{attribute 'linkalways'} 
{attribute 'no_explicit_call' := 'This FB is a CLASS and must be accessed using methods or properties'}
{attribute 'enable_dynamic_creation'}
FUNCTION_BLOCK Node_F_VN_MedianElementElementwise_TcVnPoint2_LREAL EXTENDS VisionNode
VAR
    ipContainer : _ITcVnContainer;
    aMedian : _TcVnPoint2_LREAL;
    hrPrev : _HRESULT(S_OK);
    hresult : _HRESULT(S_OK);
END_VAR

METHOD PUBLIC  Clone : I_Node
VAR
	pNode : POINTER TO Node_F_VN_MedianElementElementwise_TcVnPoint2_LREAL;
END_VAR
pNode := __NEW(Node_F_VN_MedianElementElementwise_TcVnPoint2_LREAL);
Clone := pNode^;
END_METHOD

METHOD FB_init : BOOL
VAR_INPUT
	bInitRetains : BOOL; // if TRUE, the retain variables are initialized (warm start / cold start)
	bInCopyCode : BOOL;  // if TRUE, the instance afterwards gets moved into the copy code (online change)
END_VAR
AddInput('ipContainer', ipContainer);
AddInput('aMedian', aMedian);
AddInput('hrPrev', hrPrev);
AddOutput('ipContainer', ipContainer);
AddOutput('hresult',hresult);
END_METHOD

METHOD PROTECTED OnExecute : HRESULT
hresult.Value := F_VN_MedianElementElementwise_TcVnPoint2_LREAL(
    ipContainer := ipContainer.Value,
    aMedian := aMedian.Value,
    hrPrev:= hrPrev.Value);
END_METHOD

METHOD PUBLIC PreExecutionCheck
VAR_INPUT
	Check : I_PreExecutionChecks;
END_VAR
Check.IsTrue(ipContainer.IsValid, 'ipContainer must be a valid container');
END_METHOD

END_FUNCTION_BLOCK

(* stored: Version 1.1.0.1, ProductVersion 3.1.4024.13
   POU Node_F_VN_MedianElementElementwise_TcVnPoint2_LREAL: Id {fc01a2aa-51e7-451f-8134-0c4ebfbcd398}, SpecialFunc None
   Folder Constructor: Id {32866910-878f-4bf5-b7bf-0196a97f15e1}
   Method Clone: Id {e1ed582e-0a6e-4340-971a-d9e0ecc5e0c5}
   Method FB_init: Id {cfee0542-f779-486f-a3a9-4cf7cc33ec31}
   Method OnExecute: Id {60a5be63-376b-4b96-a1fa-346e5a4276fd}
   Method PreExecutionCheck: Id {15fe0c33-115b-4e90-a28b-bcab1890b821} *)
